FUNCTION_BLOCK DiscreteTimeIntegrator_Init
VAR_INPUT
	ssMethodType: SINT;
	In: LREAL;
	Init: LREAL;
	minOut : LREAL;
	maxOut : LREAL;
	tCycle : LREAL;
END_VAR
VAR_OUTPUT
	Out: LREAL;
END_VAR
VAR
	c_DiscreteTimeIntegrator_IC: USINT;
	c_DiscreteTimeIntegrator_DS: LREAL;
END_VAR



CASE ssMethodType OF
    0: 

        c_DiscreteTimeIntegrator_IC := 1;

    1: 

        IF c_DiscreteTimeIntegrator_IC <> 0 THEN 
            c_DiscreteTimeIntegrator_DS := Init;

            IF c_DiscreteTimeIntegrator_DS >= maxOut THEN 
                c_DiscreteTimeIntegrator_DS := maxOut;
            ELSIF c_DiscreteTimeIntegrator_DS <= minOut THEN 
                c_DiscreteTimeIntegrator_DS := minOut;
            END_IF;

        END_IF;


        IF c_DiscreteTimeIntegrator_DS >= maxOut THEN 
            c_DiscreteTimeIntegrator_DS := maxOut;
        ELSIF c_DiscreteTimeIntegrator_DS <= minOut THEN 
            c_DiscreteTimeIntegrator_DS := minOut;
        END_IF;

       
        Out := c_DiscreteTimeIntegrator_DS;
        
        c_DiscreteTimeIntegrator_IC := 0;
        c_DiscreteTimeIntegrator_DS := (tCycle * In) + c_DiscreteTimeIntegrator_DS;

        IF c_DiscreteTimeIntegrator_DS >= maxOut THEN 
            c_DiscreteTimeIntegrator_DS := maxOut;
        ELSIF c_DiscreteTimeIntegrator_DS <= minOut THEN 
            c_DiscreteTimeIntegrator_DS := minOut;
        END_IF;

END_CASE;

END_FUNCTION_BLOCK

(* stored: Version 1.1.0.1, ProductVersion 3.1.4024.9
   POU DiscreteTimeIntegrator_Init: Id {4adbae3e-24df-4455-b26a-f1991cd2862f}, SpecialFunc None *)
